INTERFACE ITF_ControlElement2 EXTENDS ITF_BaseControlElement

END_INTERFACE

(* stored: Version 1.1.0.1, ProductVersion 3.1.4024.15
   Itf ITF_ControlElement2: Id {d82c59b3-0137-47db-8ef8-95596bf3d331} *)
